PROGRAM MAIN
VAR
	bTest :BOOL := TRUE;
END_VAR

RTClock();
IF bRTCValid THEN
	NewAverage();	
	PrgMqttCom();	
	Enocean_program();
	control();
	HouseControl();
	//DataExchange();
	CurrentMeassuring();
END_IF

END_PROGRAM

(* stored: Version 1.1.0.1, ProductVersion 3.1.4024.12
   POU MAIN: Id {825d181d-7c23-4bb3-bc3d-80cb4eae9ef4}, SpecialFunc None *)
